FUNCTION_BLOCK FB_Generics
VAR_GENERIC CONSTANT
	nArraySize 	: INT := 10;
END_VAR
VAR 
	nStrArray	: ARRAY[0..nArraySize] OF STRING(255);
END_VAR

END_FUNCTION_BLOCK

(* stored: Version 1.1.0.1, ProductVersion 3.1.4026.6
   POU FB_Generics: Id {cc452132-e576-4240-83b3-0233b5204bb6}, SpecialFunc None *)
